FUNCTION_BLOCK FB_RpcContext_Probe
VAR_OUTPUT ownerTask : DINT; END_VAR

ownerTask := Tc2_System.GETCURTASKINDEXEX();

{attribute 'TcRpcEnable' := '1'}
METHOD PUBLIC ReadContext : DINT
ReadContext := Tc2_System.GETCURTASKINDEXEX();
END_METHOD

END_FUNCTION_BLOCK

(* stored: Version 1.1.0.1
   POU FB_RpcContext_Probe: Id {35ed318d-1a5c-4b8b-8a93-48d74c4ed752}
   Method ReadContext: Id {df162e03-79bd-42a4-b0af-42c0b9556496} *)
